{attribute addProperty BoxType "KL3361-0003"}
{attribute addProperty Id "Channel_1Channel_D054A87F00"}
{attribute addProperty CRC "2211813723"}
{attribute addProperty SizeInBites "0"}
{attribute addProperty SizeInBytes "0"}
TYPE KL_83D5995B :
STRUCT
	{attribute addProperty Name "Channel_1"}
	Channel_1 : Channel_D054A87F;
END_STRUCT
END_TYPE

(* stored: Version 1.2.0.0, ProductVersion 3.1.4024.9
   DUT KL_83D5995B: Id {b351e840-7d39-4317-9e3a-18bef06108cd} *)
